FUNCTION_BLOCK SC_PostPalletizer EXTENDS FB_Chain
VAR_INPUT
	bExecute : BOOL;
	bPalletizerDeliveryRequest : BOOL;
	sTLMqttName : STRING;
END_VAR
VAR_OUTPUT
	bGrantDeliveryPermission : BOOL;
END_VAR
VAR
	
	fbPalletAvailable : Sensor;
	fbRollConveyor : RollerConveyor;
	
END_VAR

SUPER^();
fbPalletAvailable();
fbRollConveyor();

METHOD PROTECTED   Busy : BOOL
VAR_INPUT
END_VAR
VAR
	stMqttPayload : ST_MqttPayload;
	messageIndex : UINT;
END_VAR
fbStepWorkerBusy();
CASE fbStepWorkerBusy.uiStep OF
	
	0: 
		THIS^.fbRollConveyor.On();
		rChainController.releaseForChain('scFirstFloor', THIS^);
		fbStepWorkerBusy.mNextStep(10);
		
	10:
		IF THIS^.fbPalletAvailable.bSignal
		THEN
			THIS^.fbRollConveyor.Off();
			fbStepWorkerBusy.mNextStep(20);
		END_IF
	
	20: 
		
		//Mqtt exchange
		IF Ads.fbMqttClient.Publish(sTLMqttName,stMqttPayload)
		THEN
			fbStepWorkerBusy.mNextStep(30);
		END_IF
	
	30:
	
		messageIndex := ADS.fbMqttClient.isNewMessage(sTLMqttName);
		IF messageIndex > 0
		THEN
			stMqttPayload := Ads.fbMqttClient.getNewMessage(messageIndex);
			fbStepWorkerBusy.mNextStep(40);
		END_IF
		
	40:
	
		THIS^.fbRollConveyor.On();
		fbStepWorkerBusy
			.mSetTimer(T#2S)
			.mNextStep(50);
			
	50:
		
		THIS^.fbRollConveyor.Off();
		Done();
		fbStepWorkerBusy.mNextStep(0);
		
END_CASE
END_METHOD

METHOD PROTECTED  Error : BOOL
VAR_INPUT
END_VAR
END_METHOD

METHOD PROTECTED  Idle : BOOL
VAR_INPUT
END_VAR
END_METHOD

METHOD PROTECTED  Init : BOOL
VAR_INPUT
END_VAR
IF ADS.fbMqttClient.Subscribe(sTopic := sTLMqttName)
THEN			
	Start();
END_IF
END_METHOD

METHOD PROTECTED  Prepare : BOOL
VAR_INPUT
END_VAR
END_METHOD

METHOD PROTECTED  Ready : BOOL
VAR_INPUT
END_VAR

fbStepWorkerReady();
CASE fbStepWorkerReady.uiStep OF
	
0:

	IF bExecute
		AND NOT fbPalletAvailable.bSignal
	THEN
		fbStepWorkerReady.mNextStep(10);
	END_IF
		
10:
	IF rChainController
		.releaseCheck(THIS^)
		.releaseFromChain(sChainReleasing := 'scFirstFloor', THIS^)
		.releaseResult(THIS^) 
	THEN
		fbStepWorkerReady.mNextStep(0);
		Execute();
	END_IF
	
END_CASE
END_METHOD

METHOD PROTECTED  Waiting : BOOL
VAR_INPUT
END_VAR
END_METHOD

END_FUNCTION_BLOCK

(* stored: Version 1.1.0.1, ProductVersion 3.1.4024.2
   POU SC_PostPalletizer: Id {d145f42d-ec17-4f04-88d0-151eae25ee5d}, SpecialFunc None
   Method Busy: Id {e4f83139-3ef9-4270-9b46-cb364ed0aa63}
   Method Error: Id {227e1a4a-9181-4c72-9758-791ceeadca23}
   Method Idle: Id {e8414480-ea7e-45a9-aa9a-1779a2dff0da}
   Method Init: Id {81442e9f-c1c0-4557-ad89-943fb77a69ab}
   Method Prepare: Id {8ab7a1a5-fb9e-4cb0-aa6f-cc8da359eb79}
   Method Ready: Id {93703002-b3cb-4109-9d67-57373c0d509a}
   Method Waiting: Id {03e2dc8c-1e89-4ce7-a1d1-0349de8fddc8} *)
